TYPE AxisDataGroup :
STRUCT
	brakeRelay AT %Q*: BOOL;        (* Set TRUE to release brake. *)
	lowLimitSwitch AT %I*: BOOL;    (* Is the low limit switch on? *)
	highLimitSwitch AT %I*: BOOL;
	lowTorque AT %I*: BOOL;         (* Is the controller in low-torque mode? *)
	controllerTemp AT %I*: UINT;    (* Controller temperature in Celsius. *)
	motorCurrent AT %I*: UINT;      (* Motor current in mA. *)
END_STRUCT
END_TYPE

(* stored: Version 1.1.0.1, ProductVersion 3.1.4022.12
   DUT AxisDataGroup: Id {42b1d3fd-52ef-4aef-92df-e912000eabc5} *)
